// TIA Portal project "利用move指令控制流水灯" (V15.1)

(* hardware
DEVICE "S7-1200 station_1"  S7-1200 Station
   slot 0: "Rack_0"  S7-1200 Rack  Rack  V1.0
   slot 1: "PLC_1"  CPU 1214C DC/DC/DC  6ES7 214-1AG40-0XB0  V4.2
DEVICE "HMI_1"  KTP700 Basic PN
   slot 0: "HMI_1"  KTP700 Basic PN  6AV2 123-2GB03-0AX0  15.1.0.0
   slot 1: "HMI_RT_1"  KTP700 Basic PN  6AV2 123-2GB03-0AX0  15.1.0.0
   slot 5: "HMI_1.IE_CP_1"  PROFINET Interface  15.0.1.0
      slot 1: "PROFINET Interface_1"  PROFINET Interface
         slot 1: "Port_1"  Port
*)

// ===== PLC "PLC_1"  CPU 1214C DC/DC/DC =====

VAR_GLOBAL   // PLC tag table "默认变量表"
   "Tag_1" AT %MD16 : Time;
   "Tag_2" AT %M0.0 : Bool;
   "Tag_3" AT %M0.1 : Bool;
   "Tag_4" AT %M4.0 : Bool;
   "Tag_5" AT %MW16 : Word;
   "Tag_6" AT %M0.2 : Bool;
   "Tag_7" AT %QW16 : Word;
END_VAR

VAR_GLOBAL   // PLC tag table "流水灯"
   "流水灯1" AT %M16.0 : Bool;
   "流水灯2" AT %M16.1 : Bool;
   "流水灯3" AT %M16.2 : Bool;
   "流水灯4" AT %M16.3 : Bool;
   "流水灯5" AT %M16.4 : Bool;
   "流水灯6" AT %M16.5 : Bool;
   "流水灯7" AT %M16.6 : Bool;
   "流水灯8" AT %M16.7 : Bool;
   "流水灯9" AT %M17.0 : Bool;
   "流水灯10" AT %M17.1 : Bool;
   "流水灯11" AT %M17.2 : Bool;
   "流水灯12" AT %M17.3 : Bool;
   "流水灯13" AT %M17.4 : Bool;
   "流水灯14" AT %M17.5 : Bool;
   "流水灯15" AT %M17.6 : Bool;
   "流水灯16" AT %M17.7 : Bool;
END_VAR

VAR_GLOBAL   // PLC tag table "流水灯1"
   "流水1" AT %Q16.0 : Bool;
   "流水2" AT %Q16.1 : Bool;
   "流水3" AT %Q16.2 : Bool;
   "流水4" AT %Q16.3 : Bool;
   "流水5" AT %Q16.4 : Bool;
   "流水6" AT %Q16.5 : Bool;
   "流水7" AT %Q16.6 : Bool;
   "流水8" AT %Q16.7 : Bool;
   "流水9" AT %Q17.0 : Bool;
   "流水10" AT %Q17.1 : Bool;
   "流水11" AT %Q17.2 : Bool;
   "流水12" AT %Q17.3 : Bool;
   "流水13" AT %Q17.4 : Bool;
   "流水14" AT %Q17.5 : Bool;
   "流水15" AT %Q17.6 : Bool;
   "流水16" AT %Q17.7 : Bool;
END_VAR

DATA_BLOCK "数据块_1"   // DB2
{ S7_Optimized_Access := 'TRUE' }
VERSION : 0.1
   VAR
      mw16 : Array[0..16] of Word;
   END_VAR
BEGIN
END_DATA_BLOCK

// folder: System blocks/Program resources

DATA_BLOCK "IEC_Timer_0_DB"   // DB1
{ S7_Optimized_Access := 'TRUE' }
AUTHOR : Simatic
FAMILY : IEC
NAME : IEC_TMR
VERSION : 1.0
// stored: InstanceOfName IEC_TIMER
"IEC_TIMER"
BEGIN
END_DATA_BLOCK

// folder: (top level)

ORGANIZATION_BLOCK "Main"   // OB1, LAD, ProgramCycle
TITLE = "Main Program Sweep (Cycle)"
{ S7_Optimized_Access := 'TRUE' }
VERSION : 0.1
   VAR_INPUT
      Initial_Call : Bool;   // Initial call of this OB
      Remanence : Bool;   // =True, if remanent data are available
   END_VAR
BEGIN

REGION Network 1: 启动停止流水灯
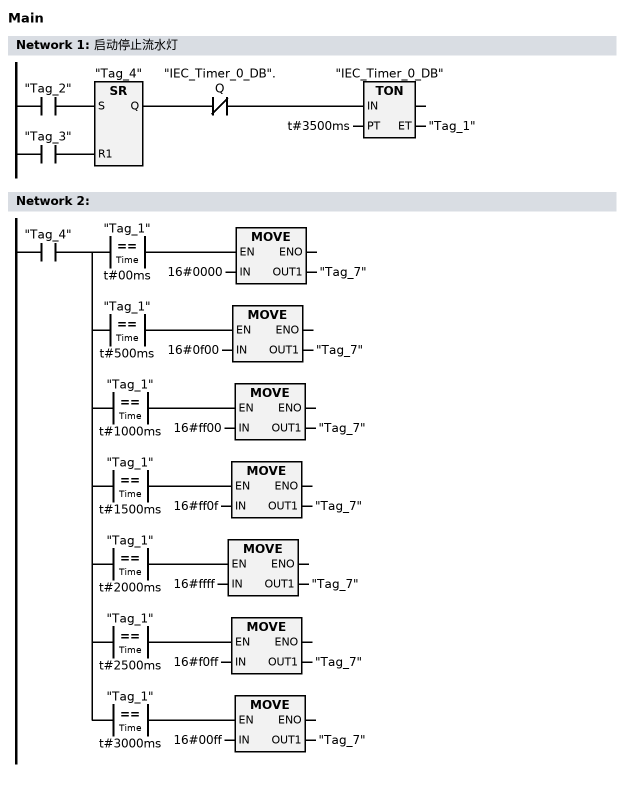
   IF "Tag_2" THEN
       "Tag_4" := TRUE;   // SR flip-flop
   END_IF;
   IF "Tag_3" THEN "Tag_4" := FALSE; END_IF;
   "IEC_Timer_0_DB".TON(IN := "Tag_4" AND NOT "IEC_Timer_0_DB".Q, PT := t#3500ms, ET => "Tag_1");
END_REGION

REGION Network 2
   RUNG wire#powerrail
      Contact( "Tag_4" )
      wire#w1
      { S7_Templates := "SrcType := Time" } EQ_Contact(in1 := "Tag_1", in2 := t#00ms)
      Move(in := 16#0000, out1 => "Tag_7")
   END_RUNG
   RUNG wire#w1
      { S7_Templates := "SrcType := Time" } EQ_Contact(in1 := "Tag_1", in2 := t#500ms)
      Move(in := 16#0f00, out1 => "Tag_7")
   END_RUNG
   RUNG wire#w1
      { S7_Templates := "SrcType := Time" } EQ_Contact(in1 := "Tag_1", in2 := t#1000ms)
      Move(in := 16#ff00, out1 => "Tag_7")
   END_RUNG
   RUNG wire#w1
      { S7_Templates := "SrcType := Time" } EQ_Contact(in1 := "Tag_1", in2 := t#1500ms)
      Move(in := 16#ff0f, out1 => "Tag_7")
   END_RUNG
   RUNG wire#w1
      { S7_Templates := "SrcType := Time" } EQ_Contact(in1 := "Tag_1", in2 := t#2000ms)
      Move(in := 16#ffff, out1 => "Tag_7")
   END_RUNG
   RUNG wire#w1
      { S7_Templates := "SrcType := Time" } EQ_Contact(in1 := "Tag_1", in2 := t#2500ms)
      Move(in := 16#f0ff, out1 => "Tag_7")
   END_RUNG
   RUNG wire#w1
      { S7_Templates := "SrcType := Time" } EQ_Contact(in1 := "Tag_1", in2 := t#3000ms)
      Move(in := 16#00ff, out1 => "Tag_7")
   END_RUNG
   // the same network as SCL:
   IF "Tag_4" AND ("Tag_1" = t#00ms) THEN "Tag_7" := 16#0000; END_IF;
   IF "Tag_4" AND ("Tag_1" = t#500ms) THEN "Tag_7" := 16#0f00; END_IF;
   IF "Tag_4" AND ("Tag_1" = t#1000ms) THEN "Tag_7" := 16#ff00; END_IF;
   IF "Tag_4" AND ("Tag_1" = t#1500ms) THEN "Tag_7" := 16#ff0f; END_IF;
   IF "Tag_4" AND ("Tag_1" = t#2000ms) THEN "Tag_7" := 16#ffff; END_IF;
   IF "Tag_4" AND ("Tag_1" = t#2500ms) THEN "Tag_7" := 16#f0ff; END_IF;
   IF "Tag_4" AND ("Tag_1" = t#3000ms) THEN "Tag_7" := 16#00ff; END_IF;
END_REGION
END_ORGANIZATION_BLOCK

(* ===== HMI "HMI_RT_1" =====
system functions are stored by id; their names below are inferred from use
connection "HMI_连接_1": ETHERNET, SMART_S7_1200_OMS

HMI tags "默认变量表"
   "Tag_ScreenNumber" : UInt, internal
   "Tag_2" : Bool = PLC Tag_2 AT %M0.0, 1 s
   "Tag_3" : Bool = PLC Tag_3 AT %M0.1, 1 s
   "流水灯1" : Bool = PLC 流水灯1 AT %M16.0, 100 ms
   "流水灯2" : Bool = PLC 流水灯2 AT %M16.1, 100 ms
   "流水灯3" : Bool = PLC 流水灯3 AT %M16.2, 100 ms
   "流水灯4" : Bool = PLC 流水灯4 AT %M16.3, 100 ms
   "流水灯5" : Bool = PLC 流水灯5 AT %M16.4, 100 ms
   "流水灯6" : Bool = PLC 流水灯6 AT %M16.5, 100 ms
   "流水灯7" : Bool = PLC 流水灯7 AT %M16.6, 100 ms
   "流水灯8" : Bool = PLC 流水灯8 AT %M16.7, 100 ms
   "流水灯9" : Bool = PLC 流水灯9 AT %M17.0, 100 ms
   "流水灯10" : Bool = PLC 流水灯10 AT %M17.1, 100 ms
   "流水灯11" : Bool = PLC 流水灯11 AT %M17.2, 100 ms
   "流水灯12" : Bool = PLC 流水灯12 AT %M17.3, 100 ms
   "流水灯13" : Bool = PLC 流水灯13 AT %M17.4, 100 ms
   "流水灯14" : Bool = PLC 流水灯14 AT %M17.5, 100 ms
   "流水灯15" : Bool = PLC 流水灯15 AT %M17.6, 100 ms
   "流水灯16" : Bool = PLC 流水灯16 AT %M17.7, 100 ms
   "流水1" : Bool = PLC 流水1 AT %Q16.0, 1 s
   "流水2" : Bool = PLC 流水2 AT %Q16.1, 1 s
   "流水3" : Bool = PLC 流水3 AT %Q16.2, 1 s
   "流水4" : Bool = PLC 流水4 AT %Q16.3, 1 s
   "流水5" : Bool = PLC 流水5 AT %Q16.4, 1 s
   "流水6" : Bool = PLC 流水6 AT %Q16.5, 1 s
   "流水7" : Bool = PLC 流水7 AT %Q16.6, 1 s
   "流水8" : Bool = PLC 流水8 AT %Q16.7, 1 s
   "流水9" : Bool = PLC 流水9 AT %Q17.0, 1 s
   "流水10" : Bool = PLC 流水10 AT %Q17.1, 1 s
   "流水11" : Bool = PLC 流水11 AT %Q17.2, 1 s
   "流水12" : Bool = PLC 流水12 AT %Q17.3, 1 s
   "流水13" : Bool = PLC 流水13 AT %Q17.4, 1 s
   "流水14" : Bool = PLC 流水14 AT %Q17.5, 1 s
   "流水15" : Bool = PLC 流水15 AT %Q17.6, 1 s
   "流水16" : Bool = PLC 流水16 AT %Q17.7, 1 s

Template "模板_1" 800x480
   Button "退出" at 714,429 size 71x50; TextOff '退出'; PictureOff "ExitRuntime_KTP700_Basic_PN_TR"; PictureOn "ExitRuntime_KTP700_Basic_PN_TR"
      on Release: StopRuntime(0)
   Button "Template_Button" at 614,429 size 71x50; TextOff 'Text'
   Button "Template_Button_1" at 514,429 size 71x50; TextOff 'Text'
   Button "Template_Button_2" at 414,429 size 71x50; TextOff 'Text'
   Button "Template_Button_3" at 314,429 size 71x50; TextOff 'Text'
   Button "Template_Button_4" at 214,429 size 71x50; TextOff 'Text'
   Button "Template_Button_5" at 114,429 size 71x50; TextOff 'Text'
   Button "起始画面" at 14,429 size 71x50; TextOff '起始画面'; PictureOff "NavigateHome_KTP700_Basic_PN_TR"; PictureOn "NavigateHome_KTP700_Basic_PN_TR"
      on Release: ActivateScreen("根画面", 0)
   SymbolicIOField "Symbolic_IO_Field_Screen" at 93,9 size 600x33; TextOff '0'; TextOn '1'; TextList "TextList_ScreenNames"
      ProcessValue <- "Tag_ScreenNumber"
      on Change: ActivateScreenByNumber("Tag_ScreenNumber", 0)
   DateTimeField "HmiScreenItemData" at 695,25 size 105x25
   DateTimeField "HmiScreenItemData_1" at 695,0 size 105x25
   GraphicView "Logo" at 0,0 size 91x51; Picture "HMI_1 的 Logo"

screen "根画面" 800x480, template "模板_1"
   on GenerateScreen: SetTag("Tag_ScreenNumber", 1)
   TextField "文本域_1" at 246,53 size 236x37; Text '控制流水灯开关'
   Rectangle "矩形_1" at 286,145 size 213x12
      Appearance <- "流水15"
   Rectangle "矩形_2" at 497,145 size 12x127
      Appearance <- "流水14"
   Rectangle "矩形_3" at 272,145 size 14x123
      Appearance <- "流水16"
   Rectangle "矩形_4" at 284,268 size 213x10
      Appearance <- "流水13"
   Rectangle "矩形_5" at 299,166 size 174x10
      Appearance <- "流水11"
   Rectangle "矩形_6" at 475,168 size 12x89
      Appearance <- "流水10"
   Rectangle "矩形_7" at 288,166 size 11x92
      Appearance <- "流水12"
   Rectangle "矩形_8" at 301,247 size 174x10
      Appearance <- "流水9"
   Rectangle "矩形_9" at 320,184 size 139x13
      Appearance <- "流水7"
   Rectangle "矩形_10" at 305,190 size 10x49
      Appearance <- "流水8"
   Rectangle "矩形_11" at 320,231 size 138x14
      Appearance <- "流水5"
   Rectangle "矩形_12" at 463,190 size 10x50
      Appearance <- "流水6"
   Rectangle "矩形_13" at 328,200 size 122x9
      Appearance <- "流水1"
   Rectangle "矩形_14" at 318,202 size 9x25
      Appearance <- "流水4"
   Rectangle "矩形_15" at 332,224 size 116x5
      Appearance <- "流水3"
   Rectangle "矩形_16" at 454,203 size 6x26
      Appearance <- "流水2"
   Button "按钮_1" at 668,239 size 96x32; TextOff '开关'
      on Press: SetBit("Tag_2")
      on Release: ResetBit("Tag_2")
   Button "按钮_2" at 665,303 size 96x32; TextOff '停止'
      on Press: SetBit("Tag_3")
      on Release: ResetBit("Tag_3")
*)